FUNCTION_BLOCK NullDigitalInputChannel implements I_DigitalInput

PROPERTY PUBLIC State : BOOL
GET
State := FALSE;
END_GET
END_PROPERTY

END_FUNCTION_BLOCK

(* stored: Version 1.1.0.1, ProductVersion 3.1.4024.5
   POU NullDigitalInputChannel: Id {fc2a3217-4cd6-4828-a534-7afe34fef2ce}, SpecialFunc None
   Property State: Id {cb8616eb-5b33-4a93-8aa7-d3f72935650d}
   Get Get: Id {158937ce-e882-48a8-9296-71b4c6edcb23} *)
